// Expose the real file request state for the cancellation test.
FUNCTION_BLOCK TestWriteStringToFile EXTENDS TOF_FileSystem.WriteString255ToFile

PROPERTY WriteBusy : BOOL
GET
WriteBusy := _PutString.bBusy;
END_GET
END_PROPERTY

END_FUNCTION_BLOCK

(* stored: Version 1.1.0.1
   POU TestWriteStringToFile: Id {234f0395-1205-4754-8e47-e2a3bcff98fe}, SpecialFunc None
   Property WriteBusy: Id {f568e06c-cbbe-4f76-9c8b-dcce163185eb}
   Get Get: Id {cc19cb3a-c6f3-4a91-b3d8-7b9b1b15013c} *)
